// TIA Portal V20 export
FUNCTION_BLOCK "Simulation"   // FB32842, LAD
// stored: MemoryReserve 100, Namespace Unit1.Em10, SetENOAutomatically false
   VAR_INPUT
      simulation { ExternalAccessible := 'False'; ExternalVisible := 'False'; ExternalWritable := 'False'} : Bool;
   END_VAR
   VAR
      instActuator { ExternalAccessible := 'False'; ExternalVisible := 'False'; ExternalWritable := 'False'} : Array[0..9] of "Simulation_Actuator";
      statDigitalSignal { ExternalAccessible := 'False'; ExternalVisible := 'False'; ExternalWritable := 'False'} : Array[0..9] of Bool;
   END_VAR
BEGIN

REGION Network 1: Digital Signal
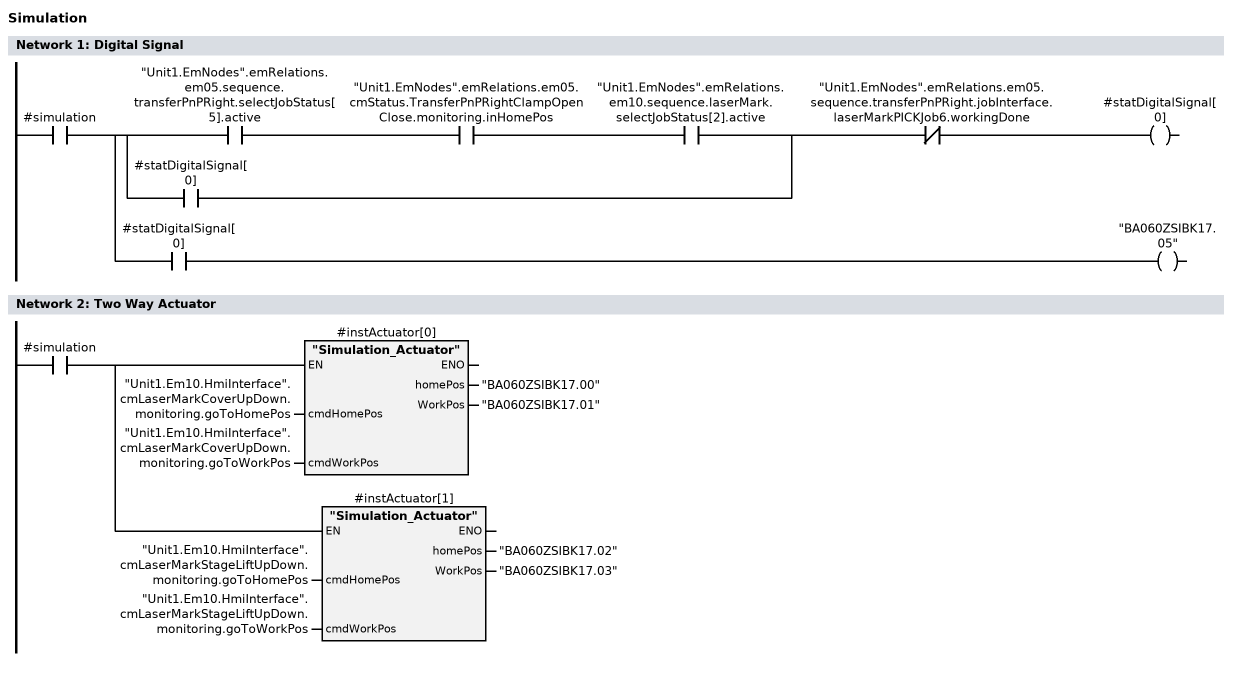
   RUNG wire#powerrail
      Contact( #simulation )
      wire#w1
      Contact( "Unit1.EmNodes".emRelations.em05.sequence.transferPnPRight.selectJobStatus[5].active )
      Contact( "Unit1.EmNodes".emRelations.em05.cmStatus.TransferPnPRightClampOpenClose.monitoring.inHomePos )
      Contact( "Unit1.EmNodes".emRelations.em10.sequence.laserMark.selectJobStatus[2].active )
      wire#w2
      I_Contact( "Unit1.EmNodes".emRelations.em05.sequence.transferPnPRight.jobInterface.laserMarkPICKJob6.workingDone )
      Coil( #statDigitalSignal[0] )
   END_RUNG
   RUNG wire#w1
      Contact( #statDigitalSignal[0] )
   END_RUNG wire#w2
   RUNG wire#w1
      Contact( #statDigitalSignal[0] )
      Coil( "BA060ZSIBK17.05" )
   END_RUNG
   // the same network as SCL:
   #statDigitalSignal[0] := #simulation AND (("Unit1.EmNodes".emRelations.em05.sequence.transferPnPRight.selectJobStatus[5].active AND "Unit1.EmNodes".emRelations.em05.cmStatus.TransferPnPRightClampOpenClose.monitoring.inHomePos AND "Unit1.EmNodes".emRelations.em10.sequence.laserMark.selectJobStatus[2].active) OR #statDigitalSignal[0]) AND NOT "Unit1.EmNodes".emRelations.em05.sequence.transferPnPRight.jobInterface.laserMarkPICKJob6.workingDone;
   "BA060ZSIBK17.05" := #simulation AND #statDigitalSignal[0];
END_REGION

REGION Network 2: Two Way Actuator
   RUNG wire#powerrail
      Contact( #simulation )
      wire#w1
      #instActuator[0](cmdHomePos := "Unit1.Em10.HmiInterface".cmLaserMarkCoverUpDown.monitoring.goToHomePos, cmdWorkPos := "Unit1.Em10.HmiInterface".cmLaserMarkCoverUpDown.monitoring.goToWorkPos, homePos => "BA060ZSIBK17.00", WorkPos => "BA060ZSIBK17.01")
   END_RUNG
   RUNG wire#w1
      #instActuator[1](cmdHomePos := "Unit1.Em10.HmiInterface".cmLaserMarkStageLiftUpDown.monitoring.goToHomePos, cmdWorkPos := "Unit1.Em10.HmiInterface".cmLaserMarkStageLiftUpDown.monitoring.goToWorkPos, homePos => "BA060ZSIBK17.02", WorkPos => "BA060ZSIBK17.03")
   END_RUNG
   // the same network as SCL:
   IF #simulation THEN
       #instActuator[0](cmdHomePos := "Unit1.Em10.HmiInterface".cmLaserMarkCoverUpDown.monitoring.goToHomePos,   // "Simulation_Actuator"
                        cmdWorkPos := "Unit1.Em10.HmiInterface".cmLaserMarkCoverUpDown.monitoring.goToWorkPos,
                        homePos => "BA060ZSIBK17.00",
                        WorkPos => "BA060ZSIBK17.01");
       #instActuator[1](cmdHomePos := "Unit1.Em10.HmiInterface".cmLaserMarkStageLiftUpDown.monitoring.goToHomePos,   // "Simulation_Actuator"
                        cmdWorkPos := "Unit1.Em10.HmiInterface".cmLaserMarkStageLiftUpDown.monitoring.goToWorkPos,
                        homePos => "BA060ZSIBK17.02",
                        WorkPos => "BA060ZSIBK17.03");
   END_IF;
END_REGION
END_FUNCTION_BLOCK
